{attribute 'linkalways'} 
{attribute 'no_explicit_call' := 'This FB is a CLASS and must be accessed using methods or properties'}
{attribute 'enable_dynamic_creation'}
FUNCTION_BLOCK _DWORD EXTENDS IntegerDatatypeBase
VAR
	localData : DWORD;
	activeData : REFERENCE TO DWORD REF= localData;
END_VAR

PROPERTY PUBLIC Address : PVOID
GET
Address := ADR(activeData);
END_GET
END_PROPERTY

METHOD PUBLIC ClearReference
VAR_INPUT
END_VAR
activeData REF= localData;
END_METHOD

METHOD PUBLIC Clone : I_Datatype
VAR
    pClone : POINTER TO _DWORD;
END_VAR
pClone := __NEW(_DWORD(InitialValue := Value));
Clone := pClone^;
END_METHOD

PROPERTY PUBLIC Datatype : T_MAXSTRING
GET
Datatype := 'DWORD';
END_GET
END_PROPERTY

METHOD FB_init : BOOL
VAR_INPUT
	bInitRetains : BOOL; // if TRUE, the retain variables are initialized (warm start / cold start)
	bInCopyCode : BOOL;  // if TRUE, the instance afterwards gets moved WORDo the copy code (online change)
	InitialValue : DWORD;
END_VAR
localData := InitialValue;
END_METHOD

PROPERTY PUBLIC IsSigned : BOOL
GET
IsSigned := FALSE;
END_GET
END_PROPERTY

PROPERTY PUBLIC LowerBound : DWORD
GET
LowerBound := DatatypeLimits.DWORD_LOWER_LIMIT;
END_GET
END_PROPERTY

METHOD PUBLIC MakeReferenceTo
VAR_INPUT
	ReferenceTarget : REFERENCE TO DWORD;
END_VAR
activeData REF= ReferenceTarget;
END_METHOD

METHOD PROTECTED SerializeLowerbound
VAR_INPUT
	Serializer : I_Serializer;
END_VAR
Serializer.AddDword(Lowerbound);
END_METHOD

METHOD PROTECTED SerializeUpperbound
VAR_INPUT
	Serializer : I_Serializer;
END_VAR
Serializer.AddDword(Upperbound);
END_METHOD

METHOD PUBLIC SerializeWith
VAR_INPUT
	Serializer : I_Serializer;
END_VAR
Serializer.AddDword(activeData);
END_METHOD

PROPERTY PUBLIC Size : UDINT
GET
Size := SIZEOF(activeData);
END_GET
END_PROPERTY

METHOD TryDeserializeFrom : BOOL
VAR_INPUT
	Deserializer : I_Deserializer;
	Feedback : I_DeserializerFeedback;
END_VAR
TryDeserializeFrom := Deserializer.TryGetDword(activeData, Feedback);
END_METHOD

METHOD TryMakeReferenceTo : BOOL
VAR_INPUT
	Target : I_Datatype;
END_VAR
VAR
	pTargetData : POINTER TO DWORD;
END_VAR
IF NOT (Target.Datatype = Datatype) THEN
	RETURN;
END_IF

pTargetData := Target.Address;
activeData REF= pTargetData^;
TryMakeReferenceTo := TRUE;
END_METHOD

PROPERTY PUBLIC UpperBound : DWORD
GET
UpperBound := DatatypeLimits.DWORD_UPPER_LIMIT;
END_GET
END_PROPERTY

PROPERTY PUBLIC Value : DWORD
GET
Value := activeData;
END_GET
SET
activeData := Value;
END_SET
END_PROPERTY

END_FUNCTION_BLOCK

(* stored: Version 1.1.0.1, ProductVersion 3.1.4024.12
   POU _DWORD: Id {e1618592-474c-06e9-0256-241d293fb756}, SpecialFunc None
   Folder Constructor: Id {6081fa35-d0fa-0615-3e40-6bcf9d5ab0f5}
   Folder Protected: Id {96d98418-62ba-0b6b-2d76-12ed5905547e}
   Property Address: Id {01b8a490-6357-09f2-2e3c-649a590225d1}
   Get Get: Id {e9fac61d-1033-05e8-074e-76511964a6c1}
   Method ClearReference: Id {2686ad7e-f5b0-0f52-0463-92f748609987}
   Method Clone: Id {bda15bdb-e191-0a8e-0b6c-fbf8237ba1f0}
   Property Datatype: Id {a92004d4-57cd-00a6-11ea-2ced8b55ecde}
   Get Get: Id {59a1ab44-0ba1-0a61-2660-8b986cb2fee7}
   Method FB_init: Id {f444b33f-03c6-0d22-0fb3-60f155eabc87}
   Property IsSigned: Id {aba69821-f124-00e4-03c3-652fd798cb58}
   Get Get: Id {2819fb0c-b977-0f9d-3668-eb598d35c185}
   Property LowerBound: Id {23c2d45a-39cd-086f-23f5-d64ddc8f4454}
   Get Get: Id {c2dd81bb-b24f-0d89-2060-a0d8ed861b35}
   Method MakeReferenceTo: Id {a1615478-51ec-04c4-0e04-7c313069d850}
   Method SerializeLowerbound: Id {4032cdcf-0b79-0a8b-1922-12cbdb2507ca}
   Method SerializeUpperbound: Id {750db5eb-be49-0cd9-0233-d973c1ca9b79}
   Method SerializeWith: Id {de88edbc-c461-0b88-0417-7a9c62325ef3}
   Property Size: Id {b30aeff7-7b0e-00a1-2cf0-7d67c573dbab}
   Get Get: Id {2c501a58-5289-0996-0022-21a91459fb34}
   Method TryDeserializeFrom: Id {6e5bd969-ed5b-05c7-106e-ef5452ab356f}
   Method TryMakeReferenceTo: Id {17213b48-96d7-0d48-04f0-2302e78f4a45}
   Property UpperBound: Id {06a0b616-9c87-0284-364a-c93d765d2559}
   Get Get: Id {b00abbe0-d40f-0845-29c0-1a45581f3768}
   Property Value: Id {d615ead0-e05e-0f6d-34dc-cb0a584b413e}
   Get Get: Id {b9f0dd16-4ed7-0445-385c-2902d495500b}
   Set Set: Id {c3676747-46e7-0cba-221a-91ced1a88394} *)
